Universal Robots PolyScope program: demo01.urp

Program demo01 (installation=default directory=/programs createdIn=5.9.1.1031110 lastSavedIn=5.9.1.1031110 robotSerialNumber=20195501059)
Calibrated DH parameters: a=[0.000146, -0.418764, -0.053981, 0.000058, -0.000023, 0]; d=[0.162545, 37.319448, -206.067439, 168.881546, 0.09955, 0.099464]; alpha=[1.57004, -0.001979, 0.002304, 1.570607, -1.57066, 0]; deltaTheta=[0, -0.174616, -1.258233, 1.432844, -0.000001, 0]
Robot Program (runOnlyOnce=true)
  MoveJ speed 60 deg/s, acceleration 80 deg/s^2 (useActiveTCP=true) feature=Base
    Waypoint Waypoint_1: TCP in base x=210.214 y=-689.207 z=159.115 mm, rx=2.2096 ry=2.1581 rz=-0.5209 rad; joints [101.88, -60.453, 82.777, -123.318, 254.213, 101.707] deg; TCP offset x=0 y=0 z=158 mm, rx=0 ry=0 rz=0 rad
  MoveL speed 250 mm/s, acceleration 1200 mm/s^2 (useActiveTCP=true) feature=Base
    Waypoint Waypoint_2: TCP in base x=19.819 y=-579.186 z=130.33 mm, rx=-2.4108 ry=-1.7684 rz=-0.0251 rad; joints [81.095, -70.063, 95.009, -108.108, 264.536, 98.912] deg
    MoveDirectionNode (selectedDirection=ZMinus toolParams=0.02, 1.2) feature=Base
      Until TOOL_CONTACT_DETECTION (allowActions=false retraction=0.002 decelerationAcceleration=3 decelerationAngularAcceleration=34.906585)
    MoveDirectionNode (selectedDirection=ZPlus) feature=Base
      Until DISTANCE (allowActions=false deceleration=3 distanceNodeType=STOP) Distance=0.02; motionParameters(blendRadius=0)
    Waypoint Waypoint_1: TCP in base x=210.214 y=-689.207 z=159.115 mm, rx=2.2096 ry=2.1581 rz=-0.5209 rad; joints [101.88, -60.453, 82.777, -123.318, 254.213, 101.707] deg
